{attribute addProperty BoxType "EM7004-0000-9995"}
{attribute addProperty Id "StatusAT %I*UINT1621ValueAT %I*UINT1622LatchAT %I*UINT1623"}
{attribute addProperty CRC "273914247"}
{attribute addProperty SizeInBites "48"}
{attribute addProperty SizeInBytes "6"}
TYPE Encoder_Channel_10539987 :
STRUCT
	{attribute addProperty Name "Status"}
	Status AT %I* : UINT;
	{attribute addProperty Name "Value"}
	Value AT %I* : UINT;
	{attribute addProperty Name "Latch"}
	Latch AT %I* : UINT;
END_STRUCT
END_TYPE

(* stored: Version 1.2.0.0, ProductVersion 3.1.4024.9
   DUT Encoder_Channel_10539987: Id {03e3c23b-89be-4700-ab35-7b9f3b1dc0b3} *)
